// TIA Portal V17 export
// export: Created 2026-07-06T15:33:04.2945123Z, ExportSetting WithDefaults, DisplayName Totally Integrated Automation Portal, DisplayVersion V17, DisplayName TIA Portal Openness, DisplayVersion V17, DisplayName TIA Portal Version Control Interface, DisplayVersion V17, DisplayName STEP 7 Professional, DisplayVersion V17, DisplayName STEP 7 Safety, DisplayVersion V17, DisplayName WinCC Professional, DisplayVersion V17
DATA_BLOCK "kinco_Data_packet_DB"   // DB9
{ S7_Optimized_Access := 'FALSE' }
VERSION : 0.1
// stored: AutoNumber true, DBAccessibleFromOPCUA true, IsOnlyStoredInLoadMemory false, IsWriteProtectedInAS false
   VAR
      Kinco_Data_Recv : Array[0..12] of Byte;
      Kinco_Data_sending_vizu : Array[0..12] of Byte;
   END_VAR
BEGIN
END_DATA_BLOCK
